// TIA Portal V16 export
// export: Created 2024-09-05T17:39:11.3023374Z, ExportSetting WithDefaults, DisplayName Totally Integrated Automation Portal, DisplayVersion V16 Update 6, DisplayName TIA Portal Version Control Interface, DisplayVersion V16 Update 2, DisplayName TIA Portal Openness, DisplayVersion V16 Update 6, DisplayName STEP 7 Professional, DisplayVersion V16 Update 6, DisplayName STEP 7 Safety, DisplayVersion V16, DisplayName WinCC Advanced, DisplayVersion V16 Update 6
DATA_BLOCK "IODiagnostic_DB"   // DB18
VERSION : 0.1
// stored: AutoNumber true, DBAccessibleFromOPCUA true, InstanceOfName IODiagnostic, InstanceOfType FB
"IODiagnostic"
   // VAR
   //    DeviceNumber : Int := 0;
   //    DeviceNumberOld : Int := 0;
   //    InputAdress : Int := 0;
   //    OutputAdress : Int := 0;
   //    InputImage : Array[1.."IOImageSize"] of Byte;
   //    OutputImage : Array[1.."IOImageSize"] of Byte;
   //    InputAdresses : Array[1.."IOImageSize"] of Int;
   //    OutputAdresses : Array[1.."IOImageSize"] of Int;
   //    SingleAdressInput : Int := 0;
   //    SingleAdressOutput : Int := 0;
   //    SingleInput : Byte := 16#06;
   //    SingleOutput : Byte := 16#00;
   //    res : Byte := 16#00;
   // END_VAR
BEGIN
   InputImage[1] := 16#06;
   InputImage[2] := 16#C0;
   InputImage[3] := 16#84;
   InputImage[4] := 16#00;
   InputImage[5] := 16#C4;
   InputImage[6] := 16#42;
   InputImage[7..14] := 16#00;
   InputImage[15] := 16#0F;
   InputImage[16..20] := 16#00;
   OutputImage[1] := 16#00;
   OutputImage[2] := 16#04;
   OutputImage[3] := 16#20;
   OutputImage[4..14] := 16#00;
   OutputImage[15] := 16#0F;
   OutputImage[16] := 16#A0;
   OutputImage[17] := 16#48;
   OutputImage[18] := 16#EE;
   OutputImage[19] := 16#14;
   OutputImage[20] := 16#00;
   InputAdresses[1] := 0;
   InputAdresses[2] := 1;
   InputAdresses[3] := 2;
   InputAdresses[4] := 3;
   InputAdresses[5] := 4;
   InputAdresses[6] := 5;
   InputAdresses[7] := 6;
   InputAdresses[8] := 7;
   InputAdresses[9] := 8;
   InputAdresses[10] := 9;
   InputAdresses[11] := 10;
   InputAdresses[12] := 11;
   InputAdresses[13] := 12;
   InputAdresses[14] := 13;
   InputAdresses[15] := 14;
   InputAdresses[16] := 15;
   InputAdresses[17] := 16;
   InputAdresses[18] := 17;
   InputAdresses[19] := 18;
   InputAdresses[20] := 19;
   OutputAdresses[1] := 0;
   OutputAdresses[2] := 1;
   OutputAdresses[3] := 2;
   OutputAdresses[4] := 3;
   OutputAdresses[5] := 4;
   OutputAdresses[6] := 5;
   OutputAdresses[7] := 6;
   OutputAdresses[8] := 7;
   OutputAdresses[9] := 8;
   OutputAdresses[10] := 9;
   OutputAdresses[11] := 10;
   OutputAdresses[12] := 11;
   OutputAdresses[13] := 12;
   OutputAdresses[14] := 13;
   OutputAdresses[15] := 14;
   OutputAdresses[16] := 15;
   OutputAdresses[17] := 16;
   OutputAdresses[18] := 17;
   OutputAdresses[19] := 18;
   OutputAdresses[20] := 19;
END_DATA_BLOCK
